FUNCTION_BLOCK FB_EstacionPreparar_SFC
VAR_INPUT
    // SFC-Flags
    SFCPause: BOOL;
    SFCReset: BOOL;
    
    // Indicadores de sincronizacion
    Benido: BOOL := TRUE;
    Ejecuta: BOOL;
    
    // Parametros
    TpoPreparacion: TIME := T#3S;
END_VAR
VAR_OUTPUT
    // Indicadores de sincronizacion
    Acabhe: BOOL;
    ListoKalisto: BOOL;
END_VAR
VAR
END_VAR

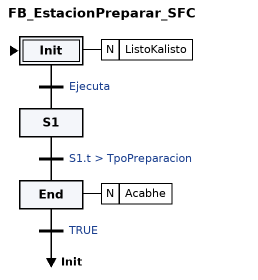
INITIAL_STEP Init:
    ListoKalisto(N);
END_STEP
TRANSITION FROM Init TO S1
    := Ejecuta;
END_TRANSITION
STEP S1:
END_STEP
TRANSITION FROM S1 TO End
    := S1.t > TpoPreparacion;
END_TRANSITION
STEP End:
    Acabhe(N);
END_STEP
TRANSITION FROM End TO Init
    := TRUE;
END_TRANSITION

END_FUNCTION_BLOCK

(* stored: Version 1.1.0.1, ProductVersion 3.1.4024.12
   POU FB_EstacionPreparar_SFC: Id {b2e6963f-6ac4-45b4-85da-9d464ae9407f}, SpecialFunc None *)
